Fanuc KAREL source: NC0019.KL

-- PROVISIONAL review KL for V770-1; original PC SHA256 96299c4f1f2194399a82e1b35c28b9e94bf49b6cc8ecc02d2ac8fa451e8a8686
-- Incomplete behavior may be omitted. Consult companion uncertainty JSON. Do not deploy.
PROGRAM NC0019
%NOLOCKGROUP
-- UNRESOLVED_LOCAL_POOL 1 cells at code offset 3; source declarations unknown
-- DIRECT_LOCAL_WORD_ACCESS alone does not prove INTEGER, REAL, or BOOLEAN
BEGIN
  -- UNRESOLVED_PC offsets 0-8; opcodes 2B,2C,7B
  -- UNRESOLVED_PC offsets 13-20; opcodes 9D,23
  -- UNRESOLVED_PC offsets 25-38; opcodes 21,9D,57,79
  -- UNRESOLVED_PC offsets 43-61; opcodes 21,2E,52,23
  -- UNRESOLVED_PC offsets 66-71; opcodes 7A
  -- UNRESOLVED_PC offsets 76-89; opcodes 21,9D,57,79
  -- UNRESOLVED_PC offsets 94-112; opcodes 21,2E,52,23
  -- UNRESOLVED_PC offsets 117-122; opcodes 7A
  -- UNRESOLVED_PC offsets 127-140; opcodes 21,9D,57,79
  -- UNRESOLVED_PC offsets 145-163; opcodes 21,2E,52,23
  -- UNRESOLVED_PC offsets 168-173; opcodes 7A
  -- UNRESOLVED_PC offsets 178-191; opcodes 21,9D,57,79
  -- UNRESOLVED_PC offsets 196-214; opcodes 21,2E,52,23
  -- UNRESOLVED_PC offsets 219-224; opcodes 7A
  -- UNRESOLVED_PC offsets 229-242; opcodes 21,9D,57,79
  -- UNRESOLVED_PC offsets 247-265; opcodes 21,2E,52,23
  -- UNRESOLVED_PC offsets 270-275; opcodes 7A
  -- UNRESOLVED_PC offsets 280-293; opcodes 21,9D,57,79
  -- UNRESOLVED_PC offsets 298-316; opcodes 21,2E,52,23
  -- UNRESOLVED_PC offsets 321-326; opcodes 7A
  -- UNRESOLVED_PC offsets 331-344; opcodes 21,9D,57,79
  -- UNRESOLVED_PC offsets 349-367; opcodes 21,2E,52,23
  -- UNRESOLVED_PC offsets 372-377; opcodes 7A
  -- UNRESOLVED_PC offsets 382-395; opcodes 21,9D,57,79
  -- UNRESOLVED_PC offsets 400-418; opcodes 21,2E,52,23
  -- UNRESOLVED_PC offsets 423-428; opcodes 7A
  -- UNRESOLVED_PC offsets 433-446; opcodes 21,9D,57,79
  -- UNRESOLVED_PC offsets 451-469; opcodes 21,2E,52,23
  -- UNRESOLVED_PC offsets 474-479; opcodes 7A
  -- UNRESOLVED_PC offsets 484-497; opcodes 21,9D,57,79
  -- UNRESOLVED_PC offsets 502-520; opcodes 21,2E,52,23
  -- UNRESOLVED_PC offsets 525-530; opcodes 7A
  -- UNRESOLVED_PC offsets 535-548; opcodes 21,9D,57,79
  -- UNRESOLVED_PC offsets 553-571; opcodes 21,2E,52,23
  -- UNRESOLVED_PC offsets 576-581; opcodes 7A
  -- UNRESOLVED_PC offsets 586-599; opcodes 21,9D,57,79
  -- UNRESOLVED_PC offsets 604-622; opcodes 21,2E,52,23
  -- UNRESOLVED_PC offsets 627-632; opcodes 7A
  -- UNRESOLVED_PC offsets 637-650; opcodes 21,9D,57,79
  -- UNRESOLVED_PC offsets 655-673; opcodes 21,2E,52,23
  -- UNRESOLVED_PC offsets 678-683; opcodes 7A
  -- UNRESOLVED_PC offsets 688-701; opcodes 21,9D,57,79
  -- UNRESOLVED_PC offsets 706-724; opcodes 21,2E,52,23
  -- UNRESOLVED_PC offsets 729-734; opcodes 7A
  -- UNRESOLVED_PC offsets 739-752; opcodes 21,9D,57,79
  -- UNRESOLVED_PC offsets 757-775; opcodes 21,2E,52,23
  -- UNRESOLVED_PC offsets 780-785; opcodes 7A
  -- UNRESOLVED_PC offsets 790-804; opcodes 21,9D,52,23
  -- UNRESOLVED_PC offsets 884-888; opcodes 7F
  -- UNRESOLVED_PC offsets 893-897; opcodes 27,AA
  -- UNRESOLVED_PC offsets 902-906; opcodes 7F
END NC0019
